// TIA Portal V19 export
// export: Created 2024-12-05T09:06:12.6435942Z, ExportSetting WithDefaults, DisplayName Totally Integrated Automation Portal, DisplayVersion V19 Update 1, DisplayName TIA Portal Openness, DisplayVersion V19 Update 1, DisplayName TIA Portal Version Control Interface, DisplayVersion V19, DisplayName SINAMICS Startdrive Advanced, DisplayVersion V19, DisplayName SINAMICS DCC, DisplayVersion V19, DisplayName SINAMICS Startdrive G130, G150, S120, S150, SINAMICS MV, G220, S200, S210, DisplayVersion V19, DisplayName SINAMICS Startdrive G110M, G120, G120C, G120D, G120P, G115D, DisplayVersion V19, DisplayName STEP 7 Professional, DisplayVersion V19 Update 1, DisplayName STEP 7 Safety, DisplayVersion V19 Update 1, DisplayName WinCC Advanced, DisplayVersion V19 Update 1, DisplayName WinCC Advanced / Unified PC, DisplayVersion V19 Update 1
DATA_BLOCK "MC1"   // DB1152
{ S7_Optimized_Access := 'TRUE' }
VERSION : 0.1
// stored: AutoNumber true, DBAccessibleFromOPCUA true, DBAccessibleFromWebserver true, InstanceOfName EM_MC, InstanceOfType UDT, IsOnlyStoredInLoadMemory false, IsWriteProtectedInAS false
"EM_MC"
   // VAR RETAIN
   //    Std : "EM_Std";
   //    Presence : "EM_MC_Presence";
   //    Param : "EM_MC_Param";
   //    LastHmiDataParam : "EM_MC_Param";
   //    Alm : "EM_MC_Alm";
   //    Sign : "EM_Sign";
   //    Input : "EM_MC_Input";
   //    Output : "EM_MC_Output";
   //    ExchangeFromChain : "EM_MC_Exchange_FromChain";
   //    ExchangeToChain : "EM_MC_Exchange_ToChain";
   //    Lamps1 : "Lamps";
   //    UpperRoller : "Roller";
   // END_VAR
BEGIN
   Std.Cfg_ModuleSync := TRUE;
   Std.Cfg_0_BelongShort_1_BelongLong := TRUE;
   Std.Cfg_0_JogWord_1_JogBit := TRUE;
   Std.AbortAlmOk := TRUE;
   Std.ServicesAbortAlmOk := TRUE;
   Std.SignOK := TRUE;
   Std.AllowCopyByCategory := TRUE;
   Std.ScOk := TRUE;
   Std.OkToStop := TRUE;
   Std.PwrDrv := TRUE;
   Std.MachineSelected := TRUE;
   Std.LocalAbortReq := FALSE;
   Std.ReqStop := FALSE;
   Std.ReqAbort := TRUE;
   Std.VisEnButtons := TRUE;
   Std.VisEnButtonsRunning := TRUE;
   Std.Ena_Suspended := TRUE;
   Std.Cfg_ModuleNumber := 3;
   Std.Cfg_InverterDiagCounter_Preset := 1;
   Std.Cfg_Num_AlmDint := 9;
   Std.Cfg_Num_SignDint := 3;
   Std.Cfg_StaPbt := 65535;
   Std.Cfg_StoPbt := 65535;
   Std.Cfg_RstPbt := -1;
   Std.Cfg_EnaPbt := 65535;
   Std.Cfg_Siren := 1;
   Std.Cfg_Stack := 1;
   Std.ModeCurrentName := 'Production';
   Std.StateCurrentName := 'Aborted';
   Std.ExchangeToGlobal.Gen.Selected := TRUE;
   Std.ExchangeToGlobal.Gen.Ena_Suspended := TRUE;
   Std.ExchangeToGlobal.Gen.sts_Stopped := FALSE;
   Std.ExchangeToGlobal.Gen.sts_Aborted := TRUE;
   Std.ExchangeToGlobal.Gen.sts_ModeAutomatic := TRUE;
   Std.ExchangeToGlobal.Gen.AxisGroupSync := TRUE;
   Std.ExchangeToGlobal.Gen.CmdMode := 1;
   Std.ExchangeToGlobal.Gen.Mode := 1;
   Std.ExchangeToGlobal.AlmOk.ThSwitch := TRUE;
   Std.ExchangeToGlobal.AlmOk.SafeComm := TRUE;
   Std.ExchangeToGlobal.AlmOk.SafeEmg := TRUE;
   Std.ExchangeToGlobal.AlmOk.SafeGuards := TRUE;
   Std.ExchangeToGlobal.AlmOk.GtaAirGroup := TRUE;
   Std.ExchangeToGlobal.AlmOk.Major := TRUE;
   Std.ExchangeToGlobal.AlmOk.Minor := TRUE;
   Std.ExchangeToGlobal.AlmOk.Spare07 := TRUE;
   Std.ExchangeToGlobal.AlmOk.Spare08 := TRUE;
   Std.ExchangeToGlobal.AlmOk.Spare09 := TRUE;
   Std.ExchangeToGlobal.AlmOk.Spare10 := TRUE;
   Std.ExchangeToGlobal.AlmOk.Spare11 := TRUE;
   Std.ExchangeToGlobal.AlmOk.Spare12 := TRUE;
   Std.ExchangeToGlobal.AlmOk.Spare13 := TRUE;
   Std.ExchangeToGlobal.AlmOk.Spare14 := TRUE;
   Std.ExchangeToGlobal.AlmOk.Spare15 := TRUE;
   Std.ExchangeToGlobal.AlmOk.Spare16 := TRUE;
   Std.ExchangeToGlobal.AlmOk.Spare17 := TRUE;
   Std.ExchangeToGlobal.AlmOk.Spare18 := TRUE;
   Std.ExchangeToGlobal.AlmOk.Spare19 := TRUE;
   Std.ExchangeToGlobal.AlmOk.Spare20 := TRUE;
   Std.ExchangeToGlobal.AlmOk.Spare21 := TRUE;
   Std.ExchangeToGlobal.AlmOk.Spare22 := TRUE;
   Std.ExchangeToGlobal.AlmOk.Spare23 := TRUE;
   Std.ExchangeToGlobal.AlmOk.Spare24 := TRUE;
   Std.ExchangeToGlobal.AlmOk.Spare25 := TRUE;
   Std.ExchangeToGlobal.AlmOk.Spare26 := TRUE;
   Std.ExchangeToGlobal.AlmOk.Spare27 := TRUE;
   Std.ExchangeToGlobal.AlmOk.Spare28 := TRUE;
   Std.ExchangeToGlobal.AlmOk.Spare29 := TRUE;
   Std.ExchangeToGlobal.AlmOk.Spare30 := TRUE;
   Std.ExchangeToGlobal.AlmOk.Spare31 := TRUE;
   Std.ExchangeToGlobal.AlmCauseOk.Ope := TRUE;
   Std.ExchangeToGlobal.AlmCauseOk.Ust := TRUE;
   Std.ExchangeToGlobal.AlmCauseOk.Dst := TRUE;
   Std.ExchangeToGlobal.AlmCauseOk.Ext := TRUE;
   Std.ExchangeToGlobal.AlmCauseOk.Mac := TRUE;
   Std.ExchangeToGlobal.AlmCauseOk.Spare05 := TRUE;
   Std.ExchangeToGlobal.AlmCauseOk.Spare06 := TRUE;
   Std.ExchangeToGlobal.AlmCauseOk.Spare07 := TRUE;
   Std.ExchangeToGlobal.AlmCauseOk.Spare08 := TRUE;
   Std.ExchangeToGlobal.AlmCauseOk.Spare09 := TRUE;
   Std.ExchangeToGlobal.AlmCauseOk.Spare10 := TRUE;
   Std.ExchangeToGlobal.AlmCauseOk.Spare11 := TRUE;
   Std.ExchangeToGlobal.AlmCauseOk.Spare12 := TRUE;
   Std.ExchangeToGlobal.AlmCauseOk.Spare13 := TRUE;
   Std.ExchangeToGlobal.AlmCauseOk.Spare14 := TRUE;
   Std.ExchangeToGlobal.AlmCauseOk.Spare15 := TRUE;
   Std.ExchangeToGlobal.AlmCauseOk.Spare16 := TRUE;
   Std.ExchangeToGlobal.AlmCauseOk.Spare17 := TRUE;
   Std.ExchangeToGlobal.AlmCauseOk.Spare18 := TRUE;
   Std.ExchangeToGlobal.AlmCauseOk.Spare19 := TRUE;
   Std.ExchangeToGlobal.AlmCauseOk.Spare20 := TRUE;
   Std.ExchangeToGlobal.AlmCauseOk.Spare21 := TRUE;
   Std.ExchangeToGlobal.AlmCauseOk.Spare22 := TRUE;
   Std.ExchangeToGlobal.AlmCauseOk.Spare23 := TRUE;
   Std.ExchangeToGlobal.AlmCauseOk.Spare24 := TRUE;
   Std.ExchangeToGlobal.AlmCauseOk.Spare25 := TRUE;
   Std.ExchangeToGlobal.AlmCauseOk.Spare26 := TRUE;
   Std.ExchangeToGlobal.AlmCauseOk.Spare27 := TRUE;
   Std.ExchangeToGlobal.AlmCauseOk.Spare28 := TRUE;
   Std.ExchangeToGlobal.AlmCauseOk.Spare29 := TRUE;
   Std.ExchangeToGlobal.AlmCauseOk.Spare30 := TRUE;
   Std.ExchangeToGlobal.AlmCauseOk.Spare31 := TRUE;
   Std.ExchangeToGlobal.AlmBannerFbk.AlmPriority := 100;
   Std.ExchangeToGlobal.AlmBannerFbk.AlmCategory := -1;
   Std.ExchangeToGlobal.AlmBannerFbk.AlmCause := -1;
   Std.ExchangeToGlobal.AlmBannerFbk.AlmID := -1;
   Std.ExchangeToGlobal.SignBannerFbk.SignPriority := 100;
   Std.ExchangeToGlobal.SignBannerFbk.SignCategory := -1;
   Std.ExchangeToGlobal.SignBannerFbk.SignID := -1;
   Std.ExchangeToGlobal.LightSiren.Cfg_StaPbt := 65535;
   Std.ExchangeToGlobal.LightSiren.Cfg_RstPbt := -1;
   Std.ExchangeToGlobal.LightSiren.Cfg_EnaPbt := 65535;
   Std.ExchangeToGlobal.LightSiren.Cfg_Siren := 1;
   Std.ExchangeToGlobal.LightSiren.Cfg_Stack := 1;
   Std.ExchangeToGlobal.PackML.Sts_Aborted := TRUE;
   Std.ExchangeToGlobal.PackML.Sts_Stopped := FALSE;
   Std.ExchangeToGlobal.PackML.Sts_AbortedEnabled := TRUE;
   Std.ExchangeToGlobal.PackML.Sts_AbortingEnabled := TRUE;
   Std.ExchangeToGlobal.PackML.Sts_ClearingEnabled := TRUE;
   Std.ExchangeToGlobal.PackML.Sts_ExecuteEnabled := TRUE;
   Std.ExchangeToGlobal.PackML.Sts_IdleEnabled := TRUE;
   Std.ExchangeToGlobal.PackML.Sts_ResettingEnabled := TRUE;
   Std.ExchangeToGlobal.PackML.Sts_StartingEnabled := TRUE;
   Std.ExchangeToGlobal.PackML.Sts_StoppedEnabled := TRUE;
   Std.ExchangeToGlobal.PackML.Sts_StoppingEnabled := TRUE;
   Std.ExchangeToGlobal.PackML.Sts_SuspendedEnabled := TRUE;
   Std.ExchangeToGlobal.PackML.Sts_SuspendingEnabled := TRUE;
   Std.ExchangeToGlobal.PackML.Sts_UnSuspendingEnabled := TRUE;
   Std.ExchangeToGlobal.SignOk := TRUE;
   Std.VisAlmTypeBool.SafeGuards := TRUE;
   Std.VisAlmTypeBool.GtaAirGroup := FALSE;
   Std.VisAlmTypeBool.Minor := FALSE;
   Std.AlmTypeOk.ThSwitch := TRUE;
   Std.AlmTypeOk.SafeComm := TRUE;
   Std.AlmTypeOk.SafeEmg := TRUE;
   Std.AlmTypeOk.SafeGuards := TRUE;
   Std.AlmTypeOk.GtaAirGroup := TRUE;
   Std.AlmTypeOk.Major := TRUE;
   Std.AlmTypeOk.Minor := TRUE;
   Std.AlmTypeOk.Spare07 := TRUE;
   Std.AlmTypeOk.Spare08 := TRUE;
   Std.AlmTypeOk.Spare09 := TRUE;
   Std.AlmTypeOk.Spare10 := TRUE;
   Std.AlmTypeOk.Spare11 := TRUE;
   Std.AlmTypeOk.Spare12 := TRUE;
   Std.AlmTypeOk.Spare13 := TRUE;
   Std.AlmTypeOk.Spare14 := TRUE;
   Std.AlmTypeOk.Spare15 := TRUE;
   Std.AlmTypeOk.Spare16 := TRUE;
   Std.AlmTypeOk.Spare17 := TRUE;
   Std.AlmTypeOk.Spare18 := TRUE;
   Std.AlmTypeOk.Spare19 := TRUE;
   Std.AlmTypeOk.Spare20 := TRUE;
   Std.AlmTypeOk.Spare21 := TRUE;
   Std.AlmTypeOk.Spare22 := TRUE;
   Std.AlmTypeOk.Spare23 := TRUE;
   Std.AlmTypeOk.Spare24 := TRUE;
   Std.AlmTypeOk.Spare25 := TRUE;
   Std.AlmTypeOk.Spare26 := TRUE;
   Std.AlmTypeOk.Spare27 := TRUE;
   Std.AlmTypeOk.Spare28 := TRUE;
   Std.AlmTypeOk.Spare29 := TRUE;
   Std.AlmTypeOk.Spare30 := TRUE;
   Std.AlmTypeOk.Spare31 := TRUE;
   Std.AlmCauseOk.Ope := TRUE;
   Std.AlmCauseOk.Ust := TRUE;
   Std.AlmCauseOk.Dst := TRUE;
   Std.AlmCauseOk.Ext := TRUE;
   Std.AlmCauseOk.Mac := TRUE;
   Std.AlmCauseOk.Spare05 := TRUE;
   Std.AlmCauseOk.Spare06 := TRUE;
   Std.AlmCauseOk.Spare07 := TRUE;
   Std.AlmCauseOk.Spare08 := TRUE;
   Std.AlmCauseOk.Spare09 := TRUE;
   Std.AlmCauseOk.Spare10 := TRUE;
   Std.AlmCauseOk.Spare11 := TRUE;
   Std.AlmCauseOk.Spare12 := TRUE;
   Std.AlmCauseOk.Spare13 := TRUE;
   Std.AlmCauseOk.Spare14 := TRUE;
   Std.AlmCauseOk.Spare15 := TRUE;
   Std.AlmCauseOk.Spare16 := TRUE;
   Std.AlmCauseOk.Spare17 := TRUE;
   Std.AlmCauseOk.Spare18 := TRUE;
   Std.AlmCauseOk.Spare19 := TRUE;
   Std.AlmCauseOk.Spare20 := TRUE;
   Std.AlmCauseOk.Spare21 := TRUE;
   Std.AlmCauseOk.Spare22 := TRUE;
   Std.AlmCauseOk.Spare23 := TRUE;
   Std.AlmCauseOk.Spare24 := TRUE;
   Std.AlmCauseOk.Spare25 := TRUE;
   Std.AlmCauseOk.Spare26 := TRUE;
   Std.AlmCauseOk.Spare27 := TRUE;
   Std.AlmCauseOk.Spare28 := TRUE;
   Std.AlmCauseOk.Spare29 := TRUE;
   Std.AlmCauseOk.Spare30 := TRUE;
   Std.AlmCauseOk.Spare31 := TRUE;
   Std.ForceCategory.SafeComm := TRUE;
   Std.ForceCategory.SafeEmg := TRUE;
   Std.AlmStruct.Category[32..63] := 1;
   Std.AlmStruct.Category[64..95] := 2;
   Std.AlmStruct.Category[96..127] := 3;
   Std.AlmStruct.Category[128..159] := 4;
   Std.AlmStruct.Category[160..191] := 5;
   Std.AlmStruct.Category[192..1023] := 6;
   Std.AlmStruct.BannerPriority[32..63] := 1;
   Std.AlmStruct.BannerPriority[64..95] := 2;
   Std.AlmStruct.BannerPriority[96..127] := 3;
   Std.AlmStruct.BannerPriority[128..159] := 4;
   Std.AlmStruct.BannerPriority[160..191] := 5;
   Std.AlmStruct.BannerPriority[192..1023] := 6;
   Std.AlmStruct.Cause[0..63] := 4;
   Std.AlmStruct.Cause[128..159] := 3;
   Std.AlmStruct.Cause[160..1023] := 4;
   Std.AlmBannerFbk.AlmPriority := 100;
   Std.AlmBannerFbk.AlmCategory := -1;
   Std.AlmBannerFbk.AlmCause := -1;
   Std.AlmBannerFbk.AlmID := -1;
   Std.SignStruct.BannerPriority[0..31] := 3;
   Std.SignStruct.BannerPriority[32..63] := 1;
   Std.SignStruct.BannerPriority[64..95] := 2;
   Std.SignBannerFbk.SignPriority := 100;
   Std.SignBannerFbk.SignCategory := -1;
   Std.SignBannerFbk.SignID := -1;
   Std.MaintenanceInput.Clock_1Hz := TRUE;
   Std.MaintenanceInput.CondToBeActivated := TRUE;
   Std.LightSiren.Cfg_StaPbt := 65535;
   Std.LightSiren.Cfg_RstPbt := -1;
   Std.LightSiren.Cfg_EnaPbt := 65535;
   Std.LightSiren.Cfg_Siren := 1;
   Std.LightSiren.Cfg_Stack := 1;
   Std.MachineStateModel.Cmd_Mode := 1;
   Std.MachineStateModel.Cmd_ModeProduce := TRUE;
   Std.MachineStateModel.Sts_StateCurrent := 9;
   Std.MachineStateModel.Sts_ModeCurrent := 1;
   Std.MachineStateModel.Sts_DisabledStates := 203776;
   Std.MachineStateModel.Sts_ProductionModeCurrent := TRUE;
   Std.MachineStateModel.Sts_ClearingEnabled := TRUE;
   Std.MachineStateModel.Sts_StoppedEnabled := TRUE;
   Std.MachineStateModel.Sts_StartingEnabled := TRUE;
   Std.MachineStateModel.Sts_IdleEnabled := TRUE;
   Std.MachineStateModel.Sts_SuspendedEnabled := TRUE;
   Std.MachineStateModel.Sts_ExecuteEnabled := TRUE;
   Std.MachineStateModel.Sts_StoppingEnabled := TRUE;
   Std.MachineStateModel.Sts_AbortingEnabled := TRUE;
   Std.MachineStateModel.Sts_AbortedEnabled := TRUE;
   Std.MachineStateModel.Sts_SuspendingEnabled := TRUE;
   Std.MachineStateModel.Sts_UnSuspendingEnabled := TRUE;
   Std.MachineStateModel.Sts_ResettingEnabled := TRUE;
   Std.MachineStateModel.Sts_Stopped := FALSE;
   Std.MachineStateModel.Sts_Aborted := TRUE;
   Std.TON_SafetyOn.PT := T#1S;
   Std.TON_SafetyOn.IN := TRUE;
   Std.TOF_SirenEna.PT := T#5S;
   Std.TOF_SirenEna.ET := T#5S;
   Presence.Lamps1 := TRUE;
   // Alm.ThSwitch."0" : MC1.Alm.ThSwitch.0
   // Alm.ThSwitch."1" : MC1.Alm.ThSwitch.1
   // Alm.ThSwitch."2" : MC1.Alm.ThSwitch.2
   // Alm.ThSwitch."3" : MC1.Alm.ThSwitch.3
   // Alm.ThSwitch."4" : MC1.Alm.ThSwitch.4
   // Alm.ThSwitch."5" : MC1.Alm.ThSwitch.5
   // Alm.ThSwitch."6" : MC1.Alm.ThSwitch.6
   // Alm.ThSwitch."7" : MC1.Alm.ThSwitch.7
   // Alm.ThSwitch."8" : MC1.Alm.ThSwitch.8
   // Alm.ThSwitch."9" : MC1.Alm.ThSwitch.9
   // Alm.ThSwitch."10" : MC1.Alm.ThSwitch.10
   // Alm.ThSwitch."11" : MC1.Alm.ThSwitch.11
   // Alm.ThSwitch."12" : MC1.Alm.ThSwitch.12
   // Alm.ThSwitch."13" : MC1.Alm.ThSwitch.13
   // Alm.ThSwitch."14" : MC1.Alm.ThSwitch.14
   // Alm.ThSwitch."15" : MC1.Alm.ThSwitch.15
   // Alm.ThSwitch."16" : MC1.Alm.ThSwitch.16
   // Alm.ThSwitch."17" : MC1.Alm.ThSwitch.17
   // Alm.ThSwitch."18" : MC1.Alm.ThSwitch.18
   // Alm.ThSwitch."19" : MC1.Alm.ThSwitch.19
   // Alm.ThSwitch."20" : MC1.Alm.ThSwitch.20
   // Alm.ThSwitch."21" : MC1.Alm.ThSwitch.21
   // Alm.ThSwitch."22" : MC1.Alm.ThSwitch.22
   // Alm.ThSwitch."23" : MC1.Alm.ThSwitch.23
   // Alm.ThSwitch."24" : MC1.Alm.ThSwitch.24
   // Alm.ThSwitch."25" : MC1.Alm.ThSwitch.25
   // Alm.ThSwitch."26" : MC1.Alm.ThSwitch.26
   // Alm.ThSwitch."27" : MC1.Alm.ThSwitch.27
   // Alm.ThSwitch."28" : MC1.Alm.ThSwitch.28
   // Alm.ThSwitch."29" : MC1.Alm.ThSwitch.29
   // Alm.ThSwitch."30" : MC1.Alm.ThSwitch.30
   // Alm.ThSwitch."31" : MC1.Alm.ThSwitch.31
   // Alm.SafeComm."0" : MC1.Alm.SafeComm.0 > Communication fault point IO zone MC1 (1MC300KF3)
   // Alm.SafeComm."1" : MC1.Alm.SafeComm.1
   // Alm.SafeComm."2" : MC1.Alm.SafeComm.2
   // Alm.SafeComm."3" : MC1.Alm.SafeComm.3
   // Alm.SafeComm."4" : MC1.Alm.SafeComm.4
   // Alm.SafeComm."5" : MC1.Alm.SafeComm.5
   // Alm.SafeComm."6" : MC1.Alm.SafeComm.6
   // Alm.SafeComm."7" : MC1.Alm.SafeComm.7
   // Alm.SafeComm."8" : MC1.Alm.SafeComm.8
   // Alm.SafeComm."9" : MC1.Alm.SafeComm.9
   // Alm.SafeComm."10" : MC1.Alm.SafeComm.10
   // Alm.SafeComm."11" : MC1.Alm.SafeComm.11
   // Alm.SafeComm."12" : MC1.Alm.SafeComm.12
   // Alm.SafeComm."13" : MC1.Alm.SafeComm.13
   // Alm.SafeComm."14" : MC1.Alm.SafeComm.14
   // Alm.SafeComm."15" : MC1.Alm.SafeComm.15
   // Alm.SafeComm."16" : MC1.Alm.SafeComm.16
   // Alm.SafeComm."17" : MC1.Alm.SafeComm.17
   // Alm.SafeComm."18" : MC1.Alm.SafeComm.18
   // Alm.SafeComm."19" : MC1.Alm.SafeComm.19
   // Alm.SafeComm."20" : MC1.Alm.SafeComm.20
   // Alm.SafeComm."21" : MC1.Alm.SafeComm.21
   // Alm.SafeComm."22" : MC1.Alm.SafeComm.22
   // Alm.SafeComm."23" : MC1.Alm.SafeComm.23
   // Alm.SafeComm."24" : MC1.Alm.SafeComm.24
   // Alm.SafeComm."25" : MC1.Alm.SafeComm.25
   // Alm.SafeComm."26" : MC1.Alm.SafeComm.26
   // Alm.SafeComm."27" : MC1.Alm.SafeComm.27
   // Alm.SafeComm."28" : MC1.Alm.SafeComm.28
   // Alm.SafeComm."29" : MC1.Alm.SafeComm.29
   // Alm.SafeComm."30" : MC1.Alm.SafeComm.30
   // Alm.SafeComm."31" : MC1.Alm.SafeComm.31
   // Alm.SafeEmg."0" : MC1.Alm.SafeEmg.0
   // Alm.SafeEmg."1" : MC1.Alm.SafeEmg.1
   // Alm.SafeEmg."2" : MC1.Alm.SafeEmg.2
   // Alm.SafeEmg."3" : MC1.Alm.SafeEmg.3
   // Alm.SafeEmg."4" : MC1.Alm.SafeEmg.4
   // Alm.SafeEmg."5" : MC1.Alm.SafeEmg.5
   // Alm.SafeEmg."6" : MC1.Alm.SafeEmg.6
   // Alm.SafeEmg."7" : MC1.Alm.SafeEmg.7
   // Alm.SafeEmg."8" : MC1.Alm.SafeEmg.8
   // Alm.SafeEmg."9" : MC1.Alm.SafeEmg.9
   // Alm.SafeEmg."10" : MC1.Alm.SafeEmg.10
   // Alm.SafeEmg."11" : MC1.Alm.SafeEmg.11
   // Alm.SafeEmg."12" : MC1.Alm.SafeEmg.12
   // Alm.SafeEmg."13" : MC1.Alm.SafeEmg.13
   // Alm.SafeEmg."14" : MC1.Alm.SafeEmg.14
   // Alm.SafeEmg."15" : MC1.Alm.SafeEmg.15
   // Alm.SafeEmg."16" : MC1.Alm.SafeEmg.16
   // Alm.SafeEmg."17" : MC1.Alm.SafeEmg.17
   // Alm.SafeEmg."18" : MC1.Alm.SafeEmg.18
   // Alm.SafeEmg."19" : MC1.Alm.SafeEmg.19
   // Alm.SafeEmg."20" : MC1.Alm.SafeEmg.20
   // Alm.SafeEmg."21" : MC1.Alm.SafeEmg.21
   // Alm.SafeEmg."22" : MC1.Alm.SafeEmg.22
   // Alm.SafeEmg."23" : MC1.Alm.SafeEmg.23
   // Alm.SafeEmg."24" : MC1.Alm.SafeEmg.24
   // Alm.SafeEmg."25" : MC1.Alm.SafeEmg.25
   // Alm.SafeEmg."26" : MC1.Alm.SafeEmg.26
   // Alm.SafeEmg."27" : MC1.Alm.SafeEmg.27
   // Alm.SafeEmg."28" : MC1.Alm.SafeEmg.28
   // Alm.SafeEmg."29" : MC1.Alm.SafeEmg.29
   // Alm.SafeEmg."30" : MC1.Alm.SafeEmg.30
   // Alm.SafeEmg."31" : MC1.Alm.SafeEmg.31
   // Alm.SafeGuards."0" : MC1.Alm.SafeGuards.0 > Safe guard 1 open operator side (1MC371BG2)
   // Alm.SafeGuards."1" : MC1.Alm.SafeGuards.1 > Safe guard 2 open operator side (1MC371BG4)
   // Alm.SafeGuards."2" : MC1.Alm.SafeGuards.2 > Safe guard 3 open not operator side (1MC371BG6)
   // Alm.SafeGuards."3" : MC1.Alm.SafeGuards.3 > Safe guard 4 open not operator side (1MC371BG8)
   // Alm.SafeGuards."4" : MC1.Alm.SafeGuards.4
   // Alm.SafeGuards."5" : MC1.Alm.SafeGuards.5
   // Alm.SafeGuards."6" : MC1.Alm.SafeGuards.6
   // Alm.SafeGuards."7" : MC1.Alm.SafeGuards.7
   // Alm.SafeGuards."8" : MC1.Alm.SafeGuards.8
   // Alm.SafeGuards."9" : MC1.Alm.SafeGuards.9
   // Alm.SafeGuards."10" : MC1.Alm.SafeGuards.10
   // Alm.SafeGuards."11" : MC1.Alm.SafeGuards.11
   // Alm.SafeGuards."12" : MC1.Alm.SafeGuards.12
   // Alm.SafeGuards."13" : MC1.Alm.SafeGuards.13
   // Alm.SafeGuards."14" : MC1.Alm.SafeGuards.14
   // Alm.SafeGuards."15" : MC1.Alm.SafeGuards.15
   // Alm.SafeGuards."16" : MC1.Alm.SafeGuards.16 > Module fault (1ME371KF1)
   // Alm.SafeGuards."17" : MC1.Alm.SafeGuards.17
   // Alm.SafeGuards."18" : MC1.Alm.SafeGuards.18
   // Alm.SafeGuards."19" : MC1.Alm.SafeGuards.19
   // Alm.SafeGuards."20" : MC1.Alm.SafeGuards.20
   // Alm.SafeGuards."21" : MC1.Alm.SafeGuards.21
   // Alm.SafeGuards."22" : MC1.Alm.SafeGuards.22
   // Alm.SafeGuards."23" : MC1.Alm.SafeGuards.23
   // Alm.SafeGuards."24" : MC1.Alm.SafeGuards.24
   // Alm.SafeGuards."25" : MC1.Alm.SafeGuards.25
   // Alm.SafeGuards."26" : MC1.Alm.SafeGuards.26 > Inverter upper roller fault (1MC70TB6)
   // Alm.SafeGuards."27" : MC1.Alm.SafeGuards.27
   // Alm.SafeGuards."28" : MC1.Alm.SafeGuards.28
   // Alm.SafeGuards."29" : MC1.Alm.SafeGuards.29
   // Alm.SafeGuards."30" : MC1.Alm.SafeGuards.30
   // Alm.SafeGuards."31" : MC1.Alm.SafeGuards.31
   // Alm.GtaAirGroup."0" : MC1.Alm.GtaAirGroup.0
   // Alm.GtaAirGroup."1" : MC1.Alm.GtaAirGroup.1
   // Alm.GtaAirGroup."2" : MC1.Alm.GtaAirGroup.2
   // Alm.GtaAirGroup."3" : MC1.Alm.GtaAirGroup.3
   // Alm.GtaAirGroup."4" : MC1.Alm.GtaAirGroup.4
   // Alm.GtaAirGroup."5" : MC1.Alm.GtaAirGroup.5
   // Alm.GtaAirGroup."6" : MC1.Alm.GtaAirGroup.6
   // Alm.GtaAirGroup."7" : MC1.Alm.GtaAirGroup.7
   // Alm.GtaAirGroup."8" : MC1.Alm.GtaAirGroup.8
   // Alm.GtaAirGroup."9" : MC1.Alm.GtaAirGroup.9
   // Alm.GtaAirGroup."10" : MC1.Alm.GtaAirGroup.10
   // Alm.GtaAirGroup."11" : MC1.Alm.GtaAirGroup.11
   // Alm.GtaAirGroup."12" : MC1.Alm.GtaAirGroup.12
   // Alm.GtaAirGroup."13" : MC1.Alm.GtaAirGroup.13
   // Alm.GtaAirGroup."14" : MC1.Alm.GtaAirGroup.14
   // Alm.GtaAirGroup."15" : MC1.Alm.GtaAirGroup.15
   // Alm.GtaAirGroup."16" : MC1.Alm.GtaAirGroup.16
   // Alm.GtaAirGroup."17" : MC1.Alm.GtaAirGroup.17
   // Alm.GtaAirGroup."18" : MC1.Alm.GtaAirGroup.18
   // Alm.GtaAirGroup."19" : MC1.Alm.GtaAirGroup.19
   // Alm.GtaAirGroup."20" : MC1.Alm.GtaAirGroup.20
   // Alm.GtaAirGroup."21" : MC1.Alm.GtaAirGroup.21
   // Alm.GtaAirGroup."22" : MC1.Alm.GtaAirGroup.22
   // Alm.GtaAirGroup."23" : MC1.Alm.GtaAirGroup.23
   // Alm.GtaAirGroup."24" : MC1.Alm.GtaAirGroup.24
   // Alm.GtaAirGroup."25" : MC1.Alm.GtaAirGroup.25
   // Alm.GtaAirGroup."26" : MC1.Alm.GtaAirGroup.26
   // Alm.GtaAirGroup."27" : MC1.Alm.GtaAirGroup.27
   // Alm.GtaAirGroup."28" : MC1.Alm.GtaAirGroup.28
   // Alm.GtaAirGroup."29" : MC1.Alm.GtaAirGroup.29
   // Alm.GtaAirGroup."30" : MC1.Alm.GtaAirGroup.30
   // Alm.GtaAirGroup."31" : MC1.Alm.GtaAirGroup.31
   // Alm.Major."0" : MC1.Alm.Major.0 > Instruction fault safe off inverter (1MC)
   // Alm.Major."1" : MC1.Alm.Major.1
   // Alm.Major."2" : MC1.Alm.Major.2
   // Alm.Major."3" : MC1.Alm.Major.3
   // Alm.Major."4" : MC1.Alm.Major.4
   // Alm.Major."5" : MC1.Alm.Major.5
   // Alm.Major."6" : MC1.Alm.Major.6
   // Alm.Major."7" : MC1.Alm.Major.7
   // Alm.Major."8" : MC1.Alm.Major.8
   // Alm.Major."9" : MC1.Alm.Major.9
   // Alm.Major."10" : MC1.Alm.Major.10
   // Alm.Major."11" : MC1.Alm.Major.11
   // Alm.Major."12" : MC1.Alm.Major.12
   // Alm.Major."13" : MC1.Alm.Major.13
   // Alm.Major."14" : MC1.Alm.Major.14
   // Alm.Major."15" : MC1.Alm.Major.15
   // Alm.Major."16" : MC1.Alm.Major.16
   // Alm.Major."17" : MC1.Alm.Major.17
   // Alm.Major."18" : MC1.Alm.Major.18
   // Alm.Major."19" : MC1.Alm.Major.19
   // Alm.Major."20" : MC1.Alm.Major.20
   // Alm.Major."21" : MC1.Alm.Major.21
   // Alm.Major."22" : MC1.Alm.Major.22
   // Alm.Major."23" : MC1.Alm.Major.23
   // Alm.Major."24" : MC1.Alm.Major.24
   // Alm.Major."25" : MC1.Alm.Major.25
   // Alm.Major."26" : MC1.Alm.Major.26
   // Alm.Major."27" : MC1.Alm.Major.27
   // Alm.Major."28" : MC1.Alm.Major.28
   // Alm.Major."29" : MC1.Alm.Major.29
   // Alm.Major."30" : MC1.Alm.Major.30
   // Alm.Major."31" : MC1.Alm.Major.31
   // Alm.Minor."0" : MC1.Alm.Minor.0 > Station in manual mode selected
   // Alm.Minor."1" : MC1.Alm.Minor.1
   // Alm.Minor."2" : MC1.Alm.Minor.2
   // Alm.Minor."3" : MC1.Alm.Minor.3
   // Alm.Minor."4" : MC1.Alm.Minor.4
   // Alm.Minor."5" : MC1.Alm.Minor.5
   // Alm.Minor."6" : MC1.Alm.Minor.6
   // Alm.Minor."7" : MC1.Alm.Minor.7
   // Alm.Minor."8" : MC1.Alm.Minor.8
   // Alm.Minor."9" : MC1.Alm.Minor.9
   // Alm.Minor."10" : MC1.Alm.Minor.10
   // Alm.Minor."11" : MC1.Alm.Minor.11
   // Alm.Minor."12" : MC1.Alm.Minor.12
   // Alm.Minor."13" : MC1.Alm.Minor.13
   // Alm.Minor."14" : MC1.Alm.Minor.14
   // Alm.Minor."15" : MC1.Alm.Minor.15
   // Alm.Minor."16" : MC1.Alm.Minor.16
   // Alm.Minor."17" : MC1.Alm.Minor.17
   // Alm.Minor."18" : MC1.Alm.Minor.18
   // Alm.Minor."19" : MC1.Alm.Minor.19
   // Alm.Minor."20" : MC1.Alm.Minor.20
   // Alm.Minor."21" : MC1.Alm.Minor.21
   // Alm.Minor."22" : MC1.Alm.Minor.22
   // Alm.Minor."23" : MC1.Alm.Minor.23
   // Alm.Minor."24" : MC1.Alm.Minor.24
   // Alm.Minor."25" : MC1.Alm.Minor.25
   // Alm.Minor."26" : MC1.Alm.Minor.26
   // Alm.Minor."27" : MC1.Alm.Minor.27
   // Alm.Minor."28" : MC1.Alm.Minor.28
   // Alm.Minor."29" : MC1.Alm.Minor.29
   // Alm.Minor."30" : MC1.Alm.Minor.30
   // Alm.Minor."31" : MC1.Alm.Minor.31
   // Alm.MinorLamps1."0" : MC1.Alm.MinorLamps1.0 > Lamps 1 row 1 thermal protection (1MC85QA2)
   // Alm.MinorLamps1."1" : MC1.Alm.MinorLamps1.1 > Lamps 1 row 2 thermal protection (1MC86QA2)
   // Alm.MinorLamps1."2" : MC1.Alm.MinorLamps1.2 > Lamps 1 row 3 thermal protection (1MC87QA2)
   // Alm.MinorLamps1."3" : MC1.Alm.MinorLamps1.3 > Lamps 1 row 4 thermal protection (1MC88QA2)
   // Alm.MinorLamps1."4" : MC1.Alm.MinorLamps1.4 > Lamps 1 row 5 thermal protection (1MC89QA2)
   // Alm.MinorLamps1."5" : MC1.Alm.MinorLamps1.5 > Lamps 1 row 6 thermal protection (1MC90QA2)
   // Alm.MinorLamps1."6" : MC1.Alm.MinorLamps1.6 > Lamps 1 row 7 thermal protection (1MC91QA2)
   // Alm.MinorLamps1."7" : MC1.Alm.MinorLamps1.7
   // Alm.MinorLamps1."8" : MC1.Alm.MinorLamps1.8
   // Alm.MinorLamps1."9" : MC1.Alm.MinorLamps1.9
   // Alm.MinorLamps1."10" : MC1.Alm.MinorLamps1.10 > Lamps 1 row 1 check lamp (1MC85QA3)
   // Alm.MinorLamps1."11" : MC1.Alm.MinorLamps1.11 > Lamps 1 row 2 check lamp (1MC86QA3)
   // Alm.MinorLamps1."12" : MC1.Alm.MinorLamps1.12 > Lamps 1 row 3 check lamp (1MC87QA3)
   // Alm.MinorLamps1."13" : MC1.Alm.MinorLamps1.13 > Lamps 1 row 4 check lamp (1MC88QA3)
   // Alm.MinorLamps1."14" : MC1.Alm.MinorLamps1.14 > Lamps 1 row 5 check lamp (1MC89QA3)
   // Alm.MinorLamps1."15" : MC1.Alm.MinorLamps1.15 > Lamps 1 row 6 check lamp (1MC90QA3)
   // Alm.MinorLamps1."16" : MC1.Alm.MinorLamps1.17 > Lamps 1 row 7 check lamp (1MC91QA3)
   // Alm.MinorLamps1."17" : MC1.Alm.MinorLamps1.17
   // Alm.MinorLamps1."18" : MC1.Alm.MinorLamps1.18
   // Alm.MinorLamps1."19" : MC1.Alm.MinorLamps1.19
   // Alm.MinorLamps1."20" : MC1.Alm.MinorLamps1.20 > Group lamps 1 rotation fault (1MC330BG5)
   // Alm.MinorLamps1."21" : MC1.Alm.MinorLamps1.21
   // Alm.MinorLamps1."22" : MC1.Alm.MinorLamps1.22
   // Alm.MinorLamps1."23" : MC1.Alm.MinorLamps1.23
   // Alm.MinorLamps1."24" : MC1.Alm.MinorLamps1.24
   // Alm.MinorLamps1."25" : MC1.Alm.MinorLamps1.25
   // Alm.MinorLamps1."26" : MC1.Alm.MinorLamps1.26
   // Alm.MinorLamps1."27" : MC1.Alm.MinorLamps1.27
   // Alm.MinorLamps1."28" : MC1.Alm.MinorLamps1.28
   // Alm.MinorLamps1."29" : MC1.Alm.MinorLamps1.29
   // Alm.MinorLamps1."30" : MC1.Alm.MinorLamps1.30
   // Alm.MinorLamps1."31" : MC1.Alm.MinorLamps1.31 > Timeout start condition
   // Alm.MinorRoller."0" : MC1.Alm.MinorLamps1.0 > Lamps 1 row 1 thermal protection (1MC85QA2)
   // Alm.MinorRoller."1" : MC1.Alm.MinorLamps1.1 > Lamps 1 row 2 thermal protection (1MC86QA2)
   // Alm.MinorRoller."2" : MC1.Alm.MinorLamps1.2 > Lamps 1 row 3 thermal protection (1MC87QA2)
   // Alm.MinorRoller."3" : MC1.Alm.MinorLamps1.3 > Lamps 1 row 4 thermal protection (1MC88QA2)
   // Alm.MinorRoller."4" : MC1.Alm.MinorLamps1.4 > Lamps 1 row 5 thermal protection (1MC89QA2)
   // Alm.MinorRoller."5" : MC1.Alm.MinorLamps1.5 > Lamps 1 row 6 thermal protection (1MC90QA2)
   // Alm.MinorRoller."6" : MC1.Alm.MinorLamps1.6 > Lamps 1 row 7 thermal protection (1MC91QA2)
   // Alm.MinorRoller."7" : MC1.Alm.MinorLamps1.7
   // Alm.MinorRoller."8" : MC1.Alm.MinorLamps1.8
   // Alm.MinorRoller."9" : MC1.Alm.MinorLamps1.9
   // Alm.MinorRoller."10" : MC1.Alm.MinorLamps1.10 > Lamps 1 row 1 check lamp (1MC85QA3)
   // Alm.MinorRoller."11" : MC1.Alm.MinorLamps1.11 > Lamps 1 row 2 check lamp (1MC86QA3)
   // Alm.MinorRoller."12" : MC1.Alm.MinorLamps1.12 > Lamps 1 row 3 check lamp (1MC87QA3)
   // Alm.MinorRoller."13" : MC1.Alm.MinorLamps1.13 > Lamps 1 row 4 check lamp (1MC88QA3)
   // Alm.MinorRoller."14" : MC1.Alm.MinorLamps1.14 > Lamps 1 row 5 check lamp (1MC89QA3)
   // Alm.MinorRoller."15" : MC1.Alm.MinorLamps1.15 > Lamps 1 row 6 check lamp (1MC90QA3)
   // Alm.MinorRoller."16" : MC1.Alm.MinorLamps1.17 > Lamps 1 row 7 check lamp (1MC91QA3)
   // Alm.MinorRoller."17" : MC1.Alm.MinorLamps1.17
   // Alm.MinorRoller."18" : MC1.Alm.MinorLamps1.18
   // Alm.MinorRoller."19" : MC1.Alm.MinorLamps1.19
   // Alm.MinorRoller."20" : MC1.Alm.MinorLamps1.20 > Group lamps 1 rotation fault (1MC330BG5)
   // Alm.MinorRoller."21" : MC1.Alm.MinorLamps1.21
   // Alm.MinorRoller."22" : MC1.Alm.MinorLamps1.22
   // Alm.MinorRoller."23" : MC1.Alm.MinorLamps1.23
   // Alm.MinorRoller."24" : MC1.Alm.MinorLamps1.24
   // Alm.MinorRoller."25" : MC1.Alm.MinorLamps1.25
   // Alm.MinorRoller."26" : MC1.Alm.MinorLamps1.26
   // Alm.MinorRoller."27" : MC1.Alm.MinorLamps1.27
   // Alm.MinorRoller."28" : MC1.Alm.MinorLamps1.28
   // Alm.MinorRoller."29" : MC1.Alm.MinorLamps1.29
   // Alm.MinorRoller."30" : MC1.Alm.MinorLamps1.30
   // Alm.MinorRoller."31" : MC1.Alm.MinorLamps1.31 > Timeout start condition
   // Sign.General."0" : MC1.Sign.General.0
   // Sign.General."1" : MC1.Sign.General.1
   // Sign.General."2" : MC1.Sign.General.2
   // Sign.General."3" : MC1.Sign.General.3
   // Sign.General."4" : MC1.Sign.General.4
   // Sign.General."5" : MC1.Sign.General.5
   // Sign.General."6" : MC1.Sign.General.6
   // Sign.General."7" : MC1.Sign.General.7
   // Sign.General."8" : MC1.Sign.General.8
   // Sign.General."9" : MC1.Sign.General.9
   // Sign.General."10" : MC1.Sign.General.10
   // Sign.General."11" : MC1.Sign.General.11
   // Sign.General."12" : MC1.Sign.General.12
   // Sign.General."13" : MC1.Sign.General.13
   // Sign.General."14" : MC1.Sign.General.14
   // Sign.General."15" : MC1.Sign.General.15
   // Sign.General."16" : MC1.Sign.General.16
   // Sign.General."17" : MC1.Sign.General.17
   // Sign.General."18" : MC1.Sign.General.18
   // Sign.General."19" : MC1.Sign.General.19
   // Sign.General."20" : MC1.Sign.General.20
   // Sign.General."21" : MC1.Sign.General.21
   // Sign.General."22" : MC1.Sign.General.22
   // Sign.General."23" : MC1.Sign.General.23
   // Sign.General."24" : MC1.Sign.General.24
   // Sign.General."25" : MC1.Sign.General.25
   // Sign.General."26" : MC1.Sign.General.26
   // Sign.General."27" : MC1.Sign.General.27
   // Sign.General."28" : MC1.Sign.General.28
   // Sign.General."29" : MC1.Sign.General.29
   // Sign.General."30" : MC1.Sign.General.30
   // Sign.General."31" : MC1.Sign.General.31
   // Sign.Maintenance_Req."0" : MC1.Sign.Maintenance_Req.0 > Maintenance 0 request
   // Sign.Maintenance_Req."1" : MC1.Sign.Maintenance_Req.1 > Maintenance 1 request
   // Sign.Maintenance_Req."2" : MC1.Sign.Maintenance_Req.2 > Maintenance 2 request
   // Sign.Maintenance_Req."3" : MC1.Sign.Maintenance_Req.3 > Maintenance 3 request
   // Sign.Maintenance_Req."4" : MC1.Sign.Maintenance_Req.4 > Maintenance 4 request
   // Sign.Maintenance_Req."5" : MC1.Sign.Maintenance_Req.5 > Maintenance 5 request
   // Sign.Maintenance_Req."6" : MC1.Sign.Maintenance_Req.6 > Maintenance 6 request
   // Sign.Maintenance_Req."7" : MC1.Sign.Maintenance_Req.7 > Maintenance 7 request
   // Sign.Maintenance_Req."8" : MC1.Sign.Maintenance_Req.8 > Maintenance 8 request
   // Sign.Maintenance_Req."9" : MC1.Sign.Maintenance_Req.9 > Maintenance 9 request
   // Sign.Maintenance_Req."10" : MC1.Sign.Maintenance_Req.10
   // Sign.Maintenance_Req."11" : MC1.Sign.Maintenance_Req.11
   // Sign.Maintenance_Req."12" : MC1.Sign.Maintenance_Req.12
   // Sign.Maintenance_Req."13" : MC1.Sign.Maintenance_Req.13
   // Sign.Maintenance_Req."14" : MC1.Sign.Maintenance_Req.14
   // Sign.Maintenance_Req."15" : MC1.Sign.Maintenance_Req.15
   // Sign.Maintenance_Req."16" : MC1.Sign.Maintenance_Req.16
   // Sign.Maintenance_Req."17" : MC1.Sign.Maintenance_Req.17
   // Sign.Maintenance_Req."18" : MC1.Sign.Maintenance_Req.18
   // Sign.Maintenance_Req."19" : MC1.Sign.Maintenance_Req.19
   // Sign.Maintenance_Req."20" : MC1.Sign.Maintenance_Req.20
   // Sign.Maintenance_Req."21" : MC1.Sign.Maintenance_Req.21
   // Sign.Maintenance_Req."22" : MC1.Sign.Maintenance_Req.22
   // Sign.Maintenance_Req."23" : MC1.Sign.Maintenance_Req.23
   // Sign.Maintenance_Req."24" : MC1.Sign.Maintenance_Req.24
   // Sign.Maintenance_Req."25" : MC1.Sign.Maintenance_Req.25
   // Sign.Maintenance_Req."26" : MC1.Sign.Maintenance_Req.26
   // Sign.Maintenance_Req."27" : MC1.Sign.Maintenance_Req.27
   // Sign.Maintenance_Req."28" : MC1.Sign.Maintenance_Req.28
   // Sign.Maintenance_Req."29" : MC1.Sign.Maintenance_Req.29
   // Sign.Maintenance_Req."30" : MC1.Sign.Maintenance_Req.30
   // Sign.Maintenance_Req."31" : MC1.Sign.Maintenance_Req.31
   // Sign.Maintenance_Activated."0" : MC1.Sign.Maintenance_Activated.0 > Maintenance 0 activated
   // Sign.Maintenance_Activated."1" : MC1.Sign.Maintenance_Activated.1 > Maintenance 1 activated
   // Sign.Maintenance_Activated."2" : MC1.Sign.Maintenance_Activated.2 > Maintenance 2 activated
   // Sign.Maintenance_Activated."3" : MC1.Sign.Maintenance_Activated.3 > Maintenance 3 activated
   // Sign.Maintenance_Activated."4" : MC1.Sign.Maintenance_Activated.4 > Maintenance 4 activated
   // Sign.Maintenance_Activated."5" : MC1.Sign.Maintenance_Activated.5 > Maintenance 5 activated
   // Sign.Maintenance_Activated."6" : MC1.Sign.Maintenance_Activated.6 > Maintenance 6 activated
   // Sign.Maintenance_Activated."7" : MC1.Sign.Maintenance_Activated.7 > Maintenance 7 activated
   // Sign.Maintenance_Activated."8" : MC1.Sign.Maintenance_Activated.8 > Maintenance 8 activated
   // Sign.Maintenance_Activated."9" : MC1.Sign.Maintenance_Activated.9 > Maintenance 9 activated
   // Sign.Maintenance_Activated."10" : MC1.Sign.Maintenance_Activated.10
   // Sign.Maintenance_Activated."11" : MC1.Sign.Maintenance_Activated.11
   // Sign.Maintenance_Activated."12" : MC1.Sign.Maintenance_Activated.12
   // Sign.Maintenance_Activated."13" : MC1.Sign.Maintenance_Activated.13
   // Sign.Maintenance_Activated."14" : MC1.Sign.Maintenance_Activated.14
   // Sign.Maintenance_Activated."15" : MC1.Sign.Maintenance_Activated.15
   // Sign.Maintenance_Activated."16" : MC1.Sign.Maintenance_Activated.16
   // Sign.Maintenance_Activated."17" : MC1.Sign.Maintenance_Activated.17
   // Sign.Maintenance_Activated."18" : MC1.Sign.Maintenance_Activated.18
   // Sign.Maintenance_Activated."19" : MC1.Sign.Maintenance_Activated.19
   // Sign.Maintenance_Activated."20" : MC1.Sign.Maintenance_Activated.20
   // Sign.Maintenance_Activated."21" : MC1.Sign.Maintenance_Activated.21
   // Sign.Maintenance_Activated."22" : MC1.Sign.Maintenance_Activated.22
   // Sign.Maintenance_Activated."23" : MC1.Sign.Maintenance_Activated.23
   // Sign.Maintenance_Activated."24" : MC1.Sign.Maintenance_Activated.24
   // Sign.Maintenance_Activated."25" : MC1.Sign.Maintenance_Activated.25
   // Sign.Maintenance_Activated."26" : MC1.Sign.Maintenance_Activated.26
   // Sign.Maintenance_Activated."27" : MC1.Sign.Maintenance_Activated.27
   // Sign.Maintenance_Activated."28" : MC1.Sign.Maintenance_Activated.28
   // Sign.Maintenance_Activated."29" : MC1.Sign.Maintenance_Activated.29
   // Sign.Maintenance_Activated."30" : MC1.Sign.Maintenance_Activated.30
   // Sign.Maintenance_Activated."31" : MC1.Sign.Maintenance_Activated.31
   Input.Safety.SafeZoneOk := TRUE;
   Output.ModLgh := TRUE;
   ExchangeFromChain.Chain.EnableMove := FALSE;
   ExchangeFromChain.Chain.CheckObstruction := TRUE;
   ExchangeFromChain.Chain.VMasterInPosition := TRUE;
   ExchangeFromChain.ReqWork.Lamps1 := TRUE;
   ExchangeFromChain.ReqWork.UpperRoller := TRUE;
   ExchangeToChain.OutChainObstruction.Lamps1 := TRUE;
   ExchangeToChain.OutChainObstruction.UpperRoller := TRUE;
   ExchangeToChain.AlmOKImmStopChain := TRUE;
   Lamps1.ScOk := TRUE;
   Lamps1.OkToStop := TRUE;
   Lamps1.AlmOk := TRUE;
   Lamps1.OutChainObstruction := TRUE;
   Lamps1.Input.OffMou := TRUE;
   Lamps1.Input.BrkRow2 := TRUE;
   Lamps1.Input.BrkRow3 := TRUE;
   Lamps1.Input.BrkRow4 := TRUE;
   Lamps1.Presence.Row4 := TRUE;
   Lamps1.Man.RstCmd := TRUE;
   Lamps1.Man.ScreenNumber := 303_010_301;
   Lamps1.TOF_DelayHeatingOff.PT := T#5M;
   Lamps1.TOF_DelayHeatingOff.ET := T#5M;
   Lamps1.TON_ScOk.PT := T#20S;
   Lamps1.TON_AlmRotation.PT := T#5S;
   Lamps1.TON_DelayStartCmd.PT := T#2S;
   Lamps1.TON_CheckChainStandstill.PT := T#8S;
   UpperRoller.OkToStop := TRUE;
   UpperRoller.ScOk := TRUE;
   UpperRoller.AlmOk := TRUE;
   UpperRoller.OutChainObstruction := TRUE;
   UpperRoller.Input.BrkRow := TRUE;
   UpperRoller.Input.BrkInv := TRUE;
   UpperRoller.Input.OffMou := TRUE;
   UpperRoller.Input.Inv.Rdy := TRUE;
   UpperRoller.Input.Inv.AtRef := TRUE;
   UpperRoller.Output.CmdOffMou := TRUE;
   UpperRoller.Output.Inv.Sto := TRUE;
   UpperRoller.Output.Inv.Fwd := TRUE;
   UpperRoller.Output.InvScr.Sto := TRUE;
   UpperRoller.Output.InvScr.Fwd := TRUE;
   UpperRoller.Presence.Heater := TRUE;
   UpperRoller.Man.RstCmd := TRUE;
   UpperRoller.Man.ScreenNumber := 303_020_301;
   UpperRoller.TOF_DelayReqWork.PT := T#30S;
   UpperRoller.TOF_DelayRunInvOff.PT := T#2S;
   UpperRoller.TOF_DelayRunInvOff.ET := T#2S;
   UpperRoller.TOF_DelayHeatingOff.PT := T#5M;
   UpperRoller.TOF_DelayHeatingOff.ET := T#5M;
   UpperRoller.TON_ScOk.PT := T#20S;
   UpperRoller.TON_InverterFault.PT := T#15S;
   UpperRoller.TON_AlmPos.PT := T#5S;
   UpperRoller.TON_InverterFaultScrew.PT := T#15S;
END_DATA_BLOCK
